ABB RobotStudio station: Silla.rspag

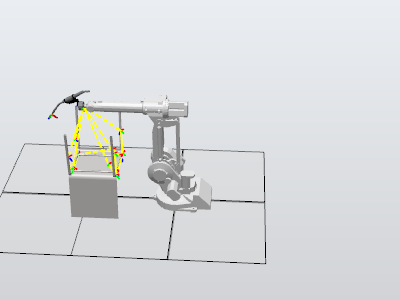
--- station ---
Station Project5 (saved by RobotStudio 23.2.10395.0)
Controller IRB1410_5_144
  mechanical unit ROB_1: IRB1410_5_144__01, 6 joints, base frame (0, 0, 0) mm
Layout (positions relative to the parent item):
  - IRB1410_5_144__01 [mechanism, from %ABB.RobotStudio.Models.IRB1410%\IRB1410_5_144_G_01.rslib] at (0, 0, 0) mm; joint values [0, 0, 0, 0, 0, 0] (rad or m)
  - AW_Gun_PSF_25 [mechanism, from %ABB.RobotStudio.Models.ArcWelding%\AW_Gun_PSF_25.rslib] at (955, 0, 1195) mm, rotated rx 0 ry 90 rz 0 deg
  - Ensamblaje1_2 [graphiccomponentgroup] at (1200, -50, 650) mm, rotated rx -90 ry 0 rz -90 deg
    - Patas:1 [part] at (-367.21, -381.14, -99.17) mm, size 600.5 x 527.8 x 22.2 mm
    - Patas:2 [part] at (-367.21, -381.14, -576.39) mm, size 600.5 x 527.8 x 22.2 mm
    - soporte1:1 [part] at (24.79, 135.6, -109.18) mm, rotated rx 0 ry 90 rz -170 deg, size 455.6 x 15.9 x 15.9 mm
    - soporte1:2 [part] at (-275.21, 135.6, -109.18) mm, rotated rx 0 ry 90 rz -170.32 deg, size 455.6 x 15.9 x 15.9 mm
    - sillla:1 [part] at (-340.3, 149.16, -337.75) mm, rotated rx 90 ry 89.87 rz -90 deg, size 520 x 540.2 x 572.6 mm
Attachment: AW_Gun_PSF_25 is attached to IRB1410_5_144__01 / Link6
Targets, tools, work objects and paths stored in the station and not in the controller backup, written as RAPID:
! task T_ROB1
MODULE CalibData
  PERS tooldata AW_Gun:=[TRUE,[[119.5,0,352],[0.890213743,0,0.455543074,0]],[1,[0,0,100],[1,0,0,0],0,0,0]];
  TASK PERS wobjdata Workobject_1:=[FALSE,TRUE,"",[[0,0,0],[1,0,0,0]],[[0,0,0],[1,0,0,0]]];
ENDMODULE

! task T_ROB1
MODULE Module1
  CONST robtarget Lado1_Inicio:=[[1115,231.943,503.292],[0.258819045,0,-0.965925826,0],[0,-1,0,0],[9E+09,9E+09,9E+09,9E+09,9E+09,9E+09]];
  CONST robtarget Lado1_Fin:=[[1115,-118.057,503.292],[0.258819045,0,-0.965925826,0],[-1,0,-1,0],[9E+09,9E+09,9E+09,9E+09,9E+09,9E+09]];
  CONST robtarget Lado1_Inicio_Ac:=[[1115,231.943,700],[0.258819045,0,-0.965925826,0],[0,-1,0,0],[9E+09,9E+09,9E+09,9E+09,9E+09,9E+09]];
  CONST robtarget Lado1_Fin_2:=[[1115,-118.057,700],[0.258819045,0,-0.965925826,0],[-1,0,-1,0],[9E+09,9E+09,9E+09,9E+09,9E+09,9E+09]];
  CONST jointtarget Home:=[[0,0,0,0,0,0],[9E+09,9E+09,9E+09,9E+09,9E+09,9E+09]];
  CONST robtarget Lado2_Inicio:=[[605,287.215,510],[0.129409523,-0.482962913,0.836516304,-0.224143868],[0,0,0,0],[9E+09,9E+09,9E+09,9E+09,9E+09,9E+09]];
  CONST robtarget Lado2_Fin:=[[605,-150,510],[0.129409523,-0.482962913,0.836516304,-0.224143868],[-1,0,-2,0],[9E+09,9E+09,9E+09,9E+09,9E+09,9E+09]];
  CONST robtarget Lado2_Inicio_Ac:=[[605,287.215,800],[0.129409523,-0.482962913,0.836516304,-0.224143868],[0,0,-1,0],[9E+09,9E+09,9E+09,9E+09,9E+09,9E+09]];
  CONST robtarget Lado2_Fin_Al:=[[605,-150,800],[0.129409523,-0.482962913,0.836516304,-0.224143868],[-1,0,-2,0],[9E+09,9E+09,9E+09,9E+09,9E+09,9E+09]];
  CONST robtarget Tubo1_Fin:=[[1090.823044184,213.88001339,507.224009294],[0.258819049,-0.000000014,0.965925825,-0.000000003],[0,0,-1,0],[9E+09,9E+09,9E+09,9E+09,9E+09,9E+09]];
  CONST robtarget Tubo1_Mitad:=[[1090.823,223.88,522.224],[0.258819046,0,0.965925826,0],[0,0,-1,0],[9E+09,9E+09,9E+09,9E+09,9E+09,9E+09]];
  CONST robtarget Tubo1_Inicio:=[[1090.823,233.88,507.224],[0.258819045,0,0.965925826,0],[0,0,0,0],[9E+09,9E+09,9E+09,9E+09,9E+09,9E+09]];
  CONST robtarget Tubo2_Inicio:=[[1090.823,-65,507.224],[0.258819045,0,0.965925826,0],[-1,-1,0,0],[9E+09,9E+09,9E+09,9E+09,9E+09,9E+09]];
  CONST robtarget Tubo2_Fin:=[[1090.823,-85,507.224],[0.258819045,0,0.965925826,0],[-1,-1,0,0],[9E+09,9E+09,9E+09,9E+09,9E+09,9E+09]];
  CONST robtarget Tubo2_Mitad:=[[1090.823,-75,522.224],[0.258819045,0,0.965925826,0],[-1,-1,0,0],[9E+09,9E+09,9E+09,9E+09,9E+09,9E+09]];
  CONST robtarget Tubo3_Inicio:=[[630,-85,507.224],[0.258819045,0,-0.965925826,0],[-1,0,-1,0],[9E+09,9E+09,9E+09,9E+09,9E+09,9E+09]];
  CONST robtarget Tubo3_Fin:=[[630,-65,507.224],[0.258819045,0,-0.965925826,0],[-1,0,-1,0],[9E+09,9E+09,9E+09,9E+09,9E+09,9E+09]];
  CONST robtarget Tubo3_Mitad:=[[630,-75,522.224],[0.258819045,0,-0.965925826,0],[-1,0,-1,0],[9E+09,9E+09,9E+09,9E+09,9E+09,9E+09]];
  CONST robtarget Intermedio:=[[700,-85,600],[0.258819045,0,-0.965925826,0],[-1,0,-1,0],[9E+09,9E+09,9E+09,9E+09,9E+09,9E+09]];
  CONST robtarget Tubo4_Inicio:=[[630,213.88,507.224],[0.258819045,0,-0.965925826,0],[0,-1,0,0],[9E+09,9E+09,9E+09,9E+09,9E+09,9E+09]];
  CONST robtarget Tubo4_Fin:=[[630,233.88,507.224],[0.258819045,0,-0.965925826,0],[0,-1,0,0],[9E+09,9E+09,9E+09,9E+09,9E+09,9E+09]];
  CONST robtarget Tubo4_Mitad:=[[630,223.88,522.224],[0.258819045,0,-0.965925826,0],[0,-1,0,0],[9E+09,9E+09,9E+09,9E+09,9E+09,9E+09]];
  CONST robtarget Ac_Inicio:=[[1080,220,550],[0.258819045,0,0.965925826,0],[0,0,-1,0],[9E+09,9E+09,9E+09,9E+09,9E+09,9E+09]];
  CONST robtarget Al_Final:=[[700,200,600],[0.258819045,0,-0.965925826,0],[0,-1,0,0],[9E+09,9E+09,9E+09,9E+09,9E+09,9E+09]];
  PROC SoldadoLado1()
    MoveAbsJ Home,v1000,z100,AW_Gun\WObj:=wobj0;
    MoveJ Lado1_Inicio_Ac,v1000,z100,AW_Gun\WObj:=wobj0;
    MoveL Lado1_Inicio,v1000,z100,AW_Gun\WObj:=wobj0;
    MoveL Lado1_Fin,v1000,z100,AW_Gun\WObj:=wobj0;
    MoveL Lado1_Fin_2,v1000,z100,AW_Gun\WObj:=wobj0;
    MoveAbsJ Home,v1000,z100,AW_Gun\WObj:=wobj0;
  ENDPROC
  PROC SoldadoLado2()
    MoveAbsJ Home,v1000,z100,AW_Gun\WObj:=wobj0;
    MoveJ Lado2_Inicio_Ac,v1000,z100,AW_Gun\WObj:=wobj0;
    MoveL Lado2_Inicio,v1000,z100,AW_Gun\WObj:=wobj0;
    MoveL Lado2_Fin,v1000,z100,AW_Gun\WObj:=wobj0;
    MoveL Lado2_Fin_Al,v1000,z100,AW_Gun\WObj:=wobj0;
    MoveAbsJ Home,v1000,z100,AW_Gun\WObj:=wobj0;
  ENDPROC
  PROC SoldadoPuntos()
    MoveAbsJ Home,v1000,z100,AW_Gun\WObj:=Workobject_1;
    MoveJ Ac_Inicio,v1000,z100,AW_Gun\WObj:=Workobject_1;
    MoveL Tubo1_Inicio,v1000,z100,AW_Gun\WObj:=Workobject_1;
    MoveL Tubo1_Mitad,v1000,z100,AW_Gun\WObj:=Workobject_1;
    MoveL Tubo1_Fin,v1000,z100,AW_Gun\WObj:=Workobject_1;
    MoveL Tubo2_Inicio,v1000,z100,AW_Gun\WObj:=Workobject_1;
    MoveL Tubo2_Mitad,v1000,z100,AW_Gun\WObj:=Workobject_1;
    MoveL Tubo2_Fin,v1000,z100,AW_Gun\WObj:=Workobject_1;
    MoveJ Intermedio,v1000,z100,AW_Gun\WObj:=Workobject_1;
    MoveL Tubo3_Inicio,v1000,z100,AW_Gun\WObj:=Workobject_1;
    MoveL Tubo3_Mitad,v1000,z100,AW_Gun\WObj:=Workobject_1;
    MoveL Tubo3_Fin,v1000,z100,AW_Gun\WObj:=Workobject_1;
    MoveL Tubo4_Inicio,v1000,z100,AW_Gun\WObj:=Workobject_1;
    MoveL Tubo4_Mitad,v1000,z100,AW_Gun\WObj:=Workobject_1;
    MoveL Tubo4_Fin,v1000,z100,AW_Gun\WObj:=Workobject_1;
    MoveL Al_Final,v1000,z100,AW_Gun\WObj:=Workobject_1;
    MoveAbsJ Home,v1000,z100,AW_Gun\WObj:=Workobject_1;
  ENDPROC
ENDMODULE


--- Controller Data/IRB1410_5_144/RAPID/TASK1/PROGMOD/Module1.mod ---
MODULE Module1
    !***********************************************************
    !
    ! M?dulo:  Module1
    !
    ! Descripción:
    !   <Introduzca la descripción aquí>
    !
    ! Autor: Andrago
    !
    ! Versión: 1.0
    !
    !***********************************************************


    !***********************************************************
    !
    ! Procedimiento Main
    !
    !   Este es el punto de entrada de su programa
    !
    !***********************************************************
    PROC main()
        !Add your code here
    ENDPROC
ENDMODULE
